(* IEC 61131-3 sources: taksa-factory-simulator/sample_programs/industrial_15/st_programs, 15 files *)

(* ---- CNCMachiningPLC10.st ---- *)
PROGRAM PLC10_CNC

VAR
    cycle_time : REAL := 120.0;
    throughput : REAL := 30.0;

    dimension_ok : BOOL := TRUE;
    surface_finish : REAL := 0.95;

    tool_break_alarm : BOOL := FALSE;

    spindle_energy : REAL := 50.0;

    machine_idle : REAL := 0.0;

    spindle_load : REAL := 70.0;
    tool_life : REAL := 100.0;

    rand : REAL;
    tick : DINT;
END_VAR

rand := REAL((tick * 41) MOD 100) / 100.0;
tick := tick + 1;

cycle_time := 100.0 + (rand * 40.0);
throughput := 3600.0 / cycle_time;

spindle_load := 60.0 + (rand * 30.0);

IF rand < 0.01 THEN
    tool_break_alarm := TRUE;
    dimension_ok := FALSE;
END_IF;

tool_life := tool_life - 0.001;

spindle_energy := spindle_load * 0.8;

END_PROGRAM

(* ---- CNCMachiningPLC8.st ---- *)
PROGRAM PLC8_CNC

VAR
    cycle_time : REAL := 120.0;
    throughput : REAL := 30.0;

    dimension_ok : BOOL := TRUE;
    surface_finish : REAL := 0.95;

    tool_break_alarm : BOOL := FALSE;

    spindle_energy : REAL := 50.0;

    machine_idle : REAL := 0.0;

    spindle_load : REAL := 70.0;
    tool_life : REAL := 100.0;

    rand : REAL;
    tick : DINT;
END_VAR

rand := REAL((tick * 41) MOD 100) / 100.0;
tick := tick + 1;

cycle_time := 100.0 + (rand * 40.0);
throughput := 3600.0 / cycle_time;

spindle_load := 60.0 + (rand * 30.0);

IF rand < 0.01 THEN
    tool_break_alarm := TRUE;
    dimension_ok := FALSE;
END_IF;

tool_life := tool_life - 0.001;

spindle_energy := spindle_load * 0.8;

END_PROGRAM

(* ---- CNCMachiningPLC9.st ---- *)
PROGRAM PLC9_CNC

VAR
    cycle_time : REAL := 120.0;
    throughput : REAL := 30.0;

    dimension_ok : BOOL := TRUE;
    surface_finish : REAL := 0.95;

    tool_break_alarm : BOOL := FALSE;

    spindle_energy : REAL := 50.0;

    machine_idle : REAL := 0.0;

    spindle_load : REAL := 70.0;
    tool_life : REAL := 100.0;

    rand : REAL;
    tick : DINT;
END_VAR

rand := REAL((tick * 41) MOD 100) / 100.0;
tick := tick + 1;

cycle_time := 100.0 + (rand * 40.0);
throughput := 3600.0 / cycle_time;

spindle_load := 60.0 + (rand * 30.0);

IF rand < 0.01 THEN
    tool_break_alarm := TRUE;
    dimension_ok := FALSE;
END_IF;

tool_life := tool_life - 0.001;

spindle_energy := spindle_load * 0.8;

END_PROGRAM

(* ---- Cooling.st ---- *)
PROGRAM PLC5_COOLING

VAR
    cooling_time : REAL := 120.0;

    cooling_uniformity : REAL := 0.95;

    temp_alarm : BOOL := FALSE;

    water_usage : REAL := 50.0;

    blockage_time : REAL := 0.0;

    pump_health : REAL := 100.0;

    rand : REAL;
    tick : DINT;
END_VAR

rand := REAL((tick * 29) MOD 100) / 100.0;
tick := tick + 1;

cooling_time := 100.0 + (rand * 40.0);
cooling_uniformity := 0.9 + (rand * 0.1);

IF rand < 0.01 THEN
    temp_alarm := TRUE;
END_IF;

water_usage := 40.0 + (rand * 20.0);

pump_health := pump_health - 0.0003;

END_PROGRAM

(* ---- Degassing.st ---- *)
PROGRAM PLC3_DEGASS

VAR
    treatment_cycle_time : REAL := 60.0;

    gas_content_level : REAL := 0.02;

    gas_leak_alarm : BOOL := FALSE;

    gas_consumption : REAL := 10.0;

    idle_time : REAL := 0.0;

    rotor_health : REAL := 100.0;

    rand : REAL;
    tick : DINT;
END_VAR

rand := REAL((tick * 19) MOD 100) / 100.0;
tick := tick + 1;

gas_content_level := 0.01 + (rand * 0.02);

IF rand < 0.005 THEN
    gas_leak_alarm := TRUE;
ELSE
    gas_leak_alarm := FALSE;
END_IF;

gas_consumption := 8.0 + (rand * 4.0);

rotor_health := rotor_health - 0.0004;

END_PROGRAM

(* ---- FinalInspection.st ---- *)
PROGRAM PLC13_FINAL_INSPECTION

VAR
    inspection_cycle : REAL := 30.0;

    crack_detected : BOOL := FALSE;
    pass_fail : BOOL := TRUE;

    radiation_alarm : BOOL := FALSE;

    energy_usage : REAL := 50.0;

    reinspection_time : REAL := 0.0;

    sensor_health : REAL := 100.0;

    rand : REAL;
    tick : DINT;
END_VAR

rand := REAL((tick * 53) MOD 100) / 100.0;
tick := tick + 1;

IF rand < 0.01 THEN
    crack_detected := TRUE;
    pass_fail := FALSE;
END_IF;

sensor_health := sensor_health - 0.0002;

END_PROGRAM

(* ---- HeatTreatment.st ---- *)
PROGRAM PLC6_HEATTREAT

VAR
    batch_cycle_time : REAL := 3600.0;

    hardness : REAL := 80.0;
    temperature_profile : REAL := 500.0;

    furnace_alarm : BOOL := FALSE;

    fuel_consumption : REAL := 300.0;

    downtime : REAL := 0.0;

    heater_health : REAL := 100.0;

    rand : REAL;
    tick : DINT;
END_VAR

rand := REAL((tick * 31) MOD 100) / 100.0;
tick := tick + 1;

temperature_profile := 480.0 + (rand * 40.0);

IF rand < 0.01 THEN
    furnace_alarm := TRUE;
END_IF;

fuel_consumption := 250.0 + (rand * 100.0);

heater_health := heater_health - 0.0004;

END_PROGRAM

(* ---- Inspection.st ---- *)
PROGRAM PLC11_INSPECTION

VAR
    inspection_rate : REAL := 60.0;

    defect_detected : BOOL := FALSE;
    defect_type : INT := 0;

    camera_fault : BOOL := FALSE;

    system_energy : REAL := 20.0;

    inspection_delay : REAL := 0.0;

    camera_health : REAL := 100.0;

    rand : REAL;
    tick : DINT;
END_VAR

rand := REAL((tick * 43) MOD 100) / 100.0;
tick := tick + 1;

IF rand < 0.02 THEN
    defect_detected := TRUE;
    defect_type := 1;
END_IF;

IF rand < 0.005 THEN
    camera_fault := TRUE;
END_IF;

camera_health := camera_health - 0.0002;

END_PROGRAM

(* ---- MeltingFurnace.st ---- *)
PROGRAM PLC2_FURNACE

VAR
    melt_rate : REAL := 100.0;
    tap_time  : REAL := 0.0;

    metal_temperature : REAL := 700.0;
    composition : REAL := 0.95;

    overheat_alarm : BOOL := FALSE;

    energy_consumption : REAL := 500.0;

    furnace_downtime : REAL := 0.0;

    refractory_health : REAL := 100.0;

    rand : REAL;
    tick : DINT;
END_VAR

rand := REAL((tick * 17) MOD 100) / 100.0;
tick := tick + 1;

// temperature control
metal_temperature := 680.0 + (rand * 50.0);

// overheat
IF metal_temperature > 720.0 THEN
    overheat_alarm := TRUE;
    furnace_downtime := furnace_downtime + 0.1;
ELSE
    overheat_alarm := FALSE;
END_IF;

melt_rate := 90.0 + (rand * 20.0);
energy_consumption := melt_rate * 4.0;

// degradation
refractory_health := refractory_health - 0.0003;

tap_time := tap_time + 0.1;

END_PROGRAM

(* ---- Packing.st ---- *)
PROGRAM PLC14_PACKING

VAR
    packing_rate : REAL := 100.0;

    packing_ok : BOOL := TRUE;

    jam_alarm : BOOL := FALSE;

    material_usage : REAL := 20.0;

    downtime : REAL := 0.0;

    robot_health : REAL := 100.0;

    rand : REAL;
    tick : DINT;
END_VAR

rand := REAL((tick * 59) MOD 100) / 100.0;
tick := tick + 1;

IF rand < 0.01 THEN
    jam_alarm := TRUE;
END_IF;

robot_health := robot_health - 0.0003;

END_PROGRAM

(* ---- Painting.st ---- *)
PROGRAM PLC12_PAINT

VAR
    coating_rate : REAL := 40.0;

    thickness : REAL := 50.0;
    finish_quality : REAL := 0.95;

    oven_alarm : BOOL := FALSE;

    powder_usage : REAL := 10.0;
    energy : REAL := 200.0;

    line_stop_time : REAL := 0.0;

    nozzle_health : REAL := 100.0;

    rand : REAL;
    tick : DINT;
END_VAR

rand := REAL((tick * 47) MOD 100) / 100.0;
tick := tick + 1;

thickness := 45.0 + (rand * 10.0);

IF rand < 0.01 THEN
    oven_alarm := TRUE;
END_IF;

nozzle_health := nozzle_health - 0.0003;

END_PROGRAM

(* ---- Press.st ---- *)
PROGRAM PLC4_PRESS

VAR
    cycle_time : REAL := 30.0;
    parts_per_hour : REAL := 100.0;

    porosity_flag : BOOL := FALSE;
    fill_quality : REAL := 0.95;

    pressure_alarm : BOOL := FALSE;

    hydraulic_energy : REAL := 200.0;

    press_idle_time : REAL := 0.0;

    press_load : REAL := 70.0;
    die_health : REAL := 100.0;

    rand : REAL;
    tick : DINT;
END_VAR

rand := REAL((tick * 23) MOD 100) / 100.0;
tick := tick + 1;

cycle_time := 25.0 + (rand * 10.0);
parts_per_hour := 3600.0 / cycle_time;

fill_quality := 0.9 + (rand * 0.1);

IF rand < 0.02 THEN
    porosity_flag := TRUE;
END_IF;

press_load := 60.0 + (rand * 30.0);

IF press_load > 85.0 THEN
    pressure_alarm := TRUE;
END_IF;

hydraulic_energy := press_load * 2.5;

die_health := die_health - 0.0005;

END_PROGRAM

(* ---- RawMaterialHandling.st ---- *)
PROGRAM PLC1_RAW_MATERIAL

VAR
    // PQSCDM
    material_feed_rate : REAL := 50.0;
    material_available : BOOL := TRUE;

    material_composition_ok : BOOL := TRUE;

    overload_alarm : BOOL := FALSE;

    energy_usage_conveyor : REAL := 5.0;

    feeder_idle_time : REAL := 0.0;

    motor_health : REAL := 100.0;

    // internal
    rand : REAL := 0.5;
    tick : DINT := 0;
END_VAR

rand := REAL((tick * 13) MOD 100) / 100.0;
tick := tick + 1;

// simulate feed variation
material_feed_rate := 45.0 + (rand * 10.0);

// occasional overload
IF rand < 0.01 THEN
    overload_alarm := TRUE;
ELSE
    overload_alarm := FALSE;
END_IF;

// idle time
IF NOT material_available THEN
    feeder_idle_time := feeder_idle_time + 0.1;
END_IF;

// degradation
motor_health := motor_health - 0.0005;

energy_usage_conveyor := material_feed_rate * 0.1;

END_PROGRAM

(* ---- ShotBlasting.st ---- *)
PROGRAM PLC7_SHOTBLAST

VAR
    cycle_time : REAL := 60.0;

    surface_cleanliness : REAL := 0.95;

    vibration_alarm : BOOL := FALSE;

    media_usage : REAL := 5.0;

    jam_time : REAL := 0.0;

    turbine_health : REAL := 100.0;

    rand : REAL;
    tick : DINT;
END_VAR

rand := REAL((tick * 37) MOD 100) / 100.0;
tick := tick + 1;

surface_cleanliness := 0.9 + (rand * 0.1);

IF rand < 0.01 THEN
    vibration_alarm := TRUE;
END_IF;

media_usage := 4.0 + (rand * 2.0);

turbine_health := turbine_health - 0.0003;

END_PROGRAM

(* ---- Utilities.st ---- *)
PROGRAM PLC15_UTILS

VAR
    supply_rate : REAL := 100.0;

    pressure_stability : REAL := 0.95;

    power_fault : BOOL := FALSE;

    total_energy : REAL := 1000.0;

    outage_time : REAL := 0.0;

    compressor_health : REAL := 100.0;

    rand : REAL;
    tick : DINT;
END_VAR

rand := REAL((tick * 61) MOD 100) / 100.0;
tick := tick + 1;

pressure_stability := 0.9 + (rand * 0.1);

IF rand < 0.005 THEN
    power_fault := TRUE;
    outage_time := outage_time + 0.1;
END_IF;

total_energy := total_energy + (rand * 10.0);

compressor_health := compressor_health - 0.0004;

END_PROGRAM
